// Mitsubishi GX Works2 project: 0716순차카운트   PLC: Q02/Q02H

// global labels: Global1
VAR_GLOBAL
  공급_후 AT X0 : BOOL;
  공급_전 AT X1 : BOOL;
  드릴_상 AT X2 : BOOL;
  드릴_하 AT X3 : BOOL;
  송출_후 AT X4 : BOOL;
  송출_전 AT X5 : BOOL;
  공솔_전 AT Y20 : BOOL;
  공솔_후 AT Y21 : BOOL;
  드릴_전 AT Y22 : BOOL;
  PB1 AT X10 : BOOL;
  PB2 AT X11 : BOOL;
END_VAR

PROGRAM MAIN
VAR
  자기_1 : 순차;
  자기_2 : 순차;
  자기_3 : 순차;
  업카_1 : 순차;
  다카_1 : 순차;
  다카_2 : 순차;
  다카_3 : 순차;
  다카_4 : 순차;
  다카_5 : 순차;
  다카_6 : 순차;
  다카_7 : 순차;
  다카_8 : 순차;
  순차_1 : 순차;
END_VAR
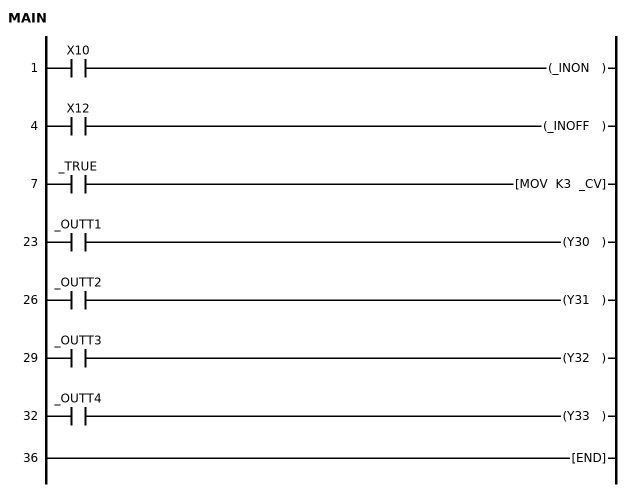
; FB BLK START 순차(순차_1)
1     LD      X10
      OUT     _INON
4     LD      X12
      OUT     _INOFF
7     LD      _TRUE
      MOV     K3 _CV
; FB START
; FB_NAME 순차
; INSTANCE_NAME 순차_1
; FB IN_B:INON
; FB OUT_OUTT1:B
; FB IN_B:INOFF
; FB OUT_OUTT2:B
; FB IN_W:CV
; FB OUT_OUTT3:B
; FB OUT_OUTT4:B
; FB END
23    LD      _OUTT1
      OUT     Y30
26    LD      _OUTT2
      OUT     Y31
29    LD      _OUTT3
      OUT     Y32
32    LD      _OUTT4
      OUT     Y33
; FB BLK END
36    END
END_PROGRAM

FUNCTION_BLOCK 순차
VAR_INPUT
  INON : BOOL;
  INOFF : BOOL;
END_VAR
VAR
  MM1 : BOOL;
  TT4 : TIMER;
  TT1 : TIMER;
  TT2 : TIMER;
  TT3 : TIMER;
END_VAR
VAR_OUTPUT
  OUTT1 : BOOL;
  OUTT2 : BOOL;
  OUTT3 : BOOL;
  OUTT4 : BOOL;
END_VAR
VAR
  CTU : COUNTER;
END_VAR
VAR_INPUT
  CV : INT;
END_VAR
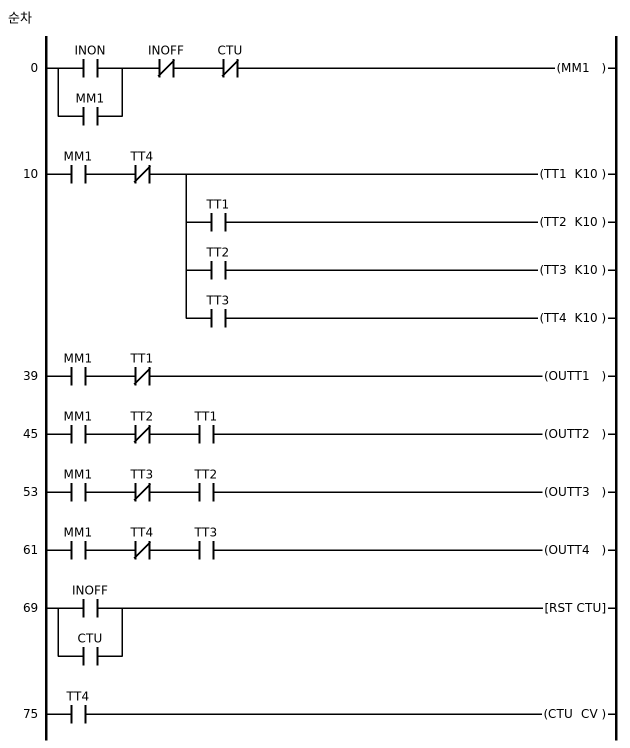
0     LD      INON
      OR      MM1
      ANI     INOFF
      ANI     CTU
      OUT     MM1
10    LD      MM1
      ANI     TT4
      OUT     TT1 K10
      MPS
      AND     TT1
      OUT     TT2 K10
      MRD
      AND     TT2
      OUT     TT3 K10
      MPP
      AND     TT3
      OUT     TT4 K10
39    LD      MM1
      ANI     TT1
      OUT     OUTT1
45    LD      MM1
      ANI     TT2
      AND     TT1
      OUT     OUTT2
53    LD      MM1
      ANI     TT3
      AND     TT2
      OUT     OUTT3
61    LD      MM1
      ANI     TT4
      AND     TT3
      OUT     OUTT4
69    LD      INOFF
      OR      CTU
      RST     CTU
75    LD      TT4
      OUT     CTU CV
END_FUNCTION_BLOCK
